PROGRAM MAIN
VAR
	robot1 : RobotLadder;
	robot2 : Robot;
	sensorBlock AT %I* : BIT8_ARRAY;
	//test : MDP5001_0_A368DC73;
END_VAR

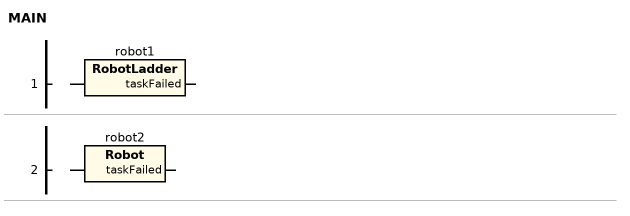
// NETWORK 1
robot1(); // RobotLadder

// NETWORK 2
robot2(); // Robot

END_PROGRAM

(* stored: Version 1.1.0.1, ProductVersion 3.1.4024.11
   POU MAIN: Id {261ae573-3319-4fbc-b33c-42387650fab7}, SpecialFunc None *)
